FUNCTION_BLOCK Cas_Stop (* Basic Function Block Type *)
  (* Standard: 61499-2 *)
  (* Version 0.2, 2003-12-04, JHC, Rockwell Automation, Renamed for better indexing. *)
  (* Version 0.1, 2002-11-05, JHC, Rockwell Automation, Corrected missing ST element in Algorithm REQ. *)
  (* Version 0.0, 2000-05-30, JHC, Rockwell Automation *)
  (* Compiler header: package fb.rt.cs725; *)
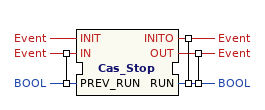
  EVENT_INPUT
    INIT; (* Initialization Request *)
    IN WITH PREV_RUN;
  END_EVENT
  EVENT_OUTPUT
    INITO WITH RUN; (* Initialization Confirm *)
    OUT WITH RUN;
  END_EVENT
  VAR_INPUT
    PREV_RUN : BOOL;
  END_VAR
  VAR_OUTPUT
    RUN : BOOL;
  END_VAR
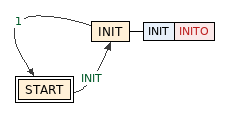
  EC_STATES
    START; (* Initial State *)
    INIT : INIT -> INITO; (* Initialization *)
  END_STATES
  EC_TRANSITIONS
    START TO INIT := INIT;
    INIT TO START := 1;
  END_TRANSITIONS
  ALGORITHM INIT IN Java: (* Initialization algorithm *)
RUN.value = true;
  END_ALGORITHM
END_FUNCTION_BLOCK
